PROGRAM TypeSizeCheck
VAR
	bundleSize : ULINT;
	adsDataSize : ULINT;
	tcpDataSize : ULINT;
	allSectionSize : ULINT;
END_VAR

bundleSize := SIZEOF(Bundle);
adsDataSize := SIZEOF(AdsData);
tcpDataSize := SIZEOF(TcpData);

allSectionSize := SIZEOF(WoodBunkEx) + SIZEOF(ChipboardEx) + SIZEOF(SpacerRecollectionUnit);

END_PROGRAM

(* stored: Version 1.1.0.1, ProductVersion 3.1.4024.11
   POU TypeSizeCheck: Id {58756afd-ee77-4842-8005-9b6b1a222eca}, SpecialFunc None *)
